PROGRAM MAIN
VAR
	fbWriteRegs : FB_WriteRegsExample;
	
END_VAR

fbWriteRegs();

END_PROGRAM

(* stored: Version 1.1.0.1, ProductVersion 3.1.4024.16
   POU MAIN: Id {251bf777-cd53-47dc-84fb-a646393ef4d0}, SpecialFunc None *)
